Universal Robots PolyScope program: timing_debug.urp

Program timing_debug (installation=timing_debug directory=/programs createdIn=5.23.0 lastSavedIn=5.23.0 robotSerialNumber=20205500786)
Calibrated DH parameters: a=[-0.000033, -0.395108, -0.391882, 0.00006, 0.000046, 0]; d=[0.16259, 52.279435, -55.760354, 3.614297, 0.099732, 0.099638]; alpha=[1.570086, -0.003008, 0.005336, 1.570553, -1.570206, 0]; deltaTheta=[0, -0.378814, 6.614643, 0.047366, 0.000002, 0.000001]
InitVariablesNode
BeforeStart
  var_4 := 4
  var_3 := 8
  var_1 := 3
  Set ExpressionOutput pin=GP_int_out[24]; expression=0
  Set ExpressionOutput pin=GP_int_out[25]; expression=0
  Set ExpressionOutput pin=GP_int_out[26]; expression=0
  Set ExpressionOutput pin=GP_int_out[27]; expression=0
  Set ExpressionOutput pin=GP_int_out[28]; expression=0
Robot Program (runOnlyOnce=false)
  Set ExpressionOutput pin=GP_int_out[28]; expression=0
  MoveJ speed 60 deg/s, acceleration 80 deg/s^2 (useActiveTCP=true optimoveEnabled=false optiMoveSpeed=0.3 optiMoveAcceleration=0.09) feature=Base
    Set ExpressionOutput pin=GP_int_out[28]; expression=GP_int_out[28]+1
    Waypoint Waypoint_1: TCP in base x=-120 y=-430 z=140 mm, rx=0 ry=3.11 rz=0.04 rad; joints [56.679, -74.282, 131.021, -144.493, -89.137, -32.909] deg
    Set ExpressionOutput pin=GP_int_out[28]; expression=GP_int_out[28]+1
    Waypoint Waypoint_2: TCP in base x=-120 y=-430 z=203.392 mm, rx=0 ry=3.11 rz=0.04 rad; joints [56.689, -82.896, 127.837, -132.695, -89.066, -32.948] deg
Thread Thread_2 (runOnlyOnce=false)
  Set ExpressionOutput pin=GP_int_out[24]; expression=0
  Set ExpressionOutput pin=GP_float_out[24]; expression=0
  var_3 := (var_3+1)%40
  If var_3≟0
    Set ExpressionOutput pin=GP_int_out[24]; expression=GP_int_out[24]+1
    tm2_s := time(2)
    'Cheap ik of the same pose'
    var_2 := get_inverse_kin(get_target_tcp_pose(), get_actual_joint_positions())
    var_2 := get_inverse_kin(get_target_tcp_pose(), get_actual_joint_positions())
    var_2 := get_inverse_kin(get_target_tcp_pose(), get_actual_joint_positions())
    var_2 := get_inverse_kin(get_target_tcp_pose(), get_actual_joint_positions())
    var_2 := get_inverse_kin(get_target_tcp_pose(), get_actual_joint_positions())
    tm2_e := time(2)
    Set ExpressionOutput pin=GP_float_out[24]; expression=(tm2_e.sec - tm2_s.sec) * 1e6 + (tm2_e.nanosec - tm2_s.nanosec) / 1e3
  Script: sync()
Thread Thread_4 (runOnlyOnce=false)
  Set ExpressionOutput pin=GP_int_out[25]; expression=0
  Set ExpressionOutput pin=GP_float_out[25]; expression=0
  var_4 := (var_4+1)%15
  If var_4≟0
    Set ExpressionOutput pin=GP_int_out[25]; expression=GP_int_out[25]+1
    tm1_s := time(2)
    'Expensive ik of different poses'
    var_2 := get_inverse_kin(get_target_tcp_pose(), get_actual_joint_positions())
    var_2 := get_inverse_kin(pose_trans(get_target_tcp_pose(), p[0.01, 0, 0, 0, 0, 0]), get_actual_joint_positions())
    var_2 := get_inverse_kin(pose_trans(get_target_tcp_pose(), p[0.02, 0, 0, 0, 0, 0]), get_actual_joint_positions())
    var_2 := get_inverse_kin(pose_trans(get_target_tcp_pose(), p[0.03, 0, 0, 0, 0, 0]), get_actual_joint_positions())
    var_2 := get_inverse_kin(pose_trans(get_target_tcp_pose(), p[0.04, 0, 0, 0, 0, 0]), get_actual_joint_positions())
    tm1_e := time(2)
    Set ExpressionOutput pin=GP_float_out[25]; expression=(tm1_e.sec - tm1_s.sec) * 1e6 + (tm1_e.nanosec - tm1_s.nanosec) / 1e3
  Script: sync()
Thread Thread_1 (runOnlyOnce=false)
  Set ExpressionOutput pin=GP_int_out[26]; expression=0
  var_1 := (var_1+1)%20
  If var_1≟0
    Set ExpressionOutput pin=GP_int_out[26]; expression=GP_int_out[26]+1
    var_2 := get_inverse_kin(get_target_tcp_pose(), get_actual_joint_positions())
  Script: sync()
Thread Thread_3 (runOnlyOnce=false)
  Set ExpressionOutput pin=GP_int_out[27]; expression=GP_int_out[27]+1
  Script: sync()
